FUNCTION_BLOCK AGVController (* Tamplate for a simple Basic Function Block Type *)
  (* Standard: 61499-2 *)
  (* Version 0.0, 2018-06-08, 4DIAC-IDE, 4DIAC-Consortium *)
  (* Version 1.0, 2016-05-26, AZ, fortiss GmbH *)
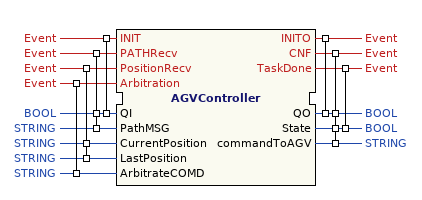
  EVENT_INPUT
    INIT WITH QI; (* Initialization Request *)
    PATHRecv WITH QI, PathMSG; (* Normal Execution Request *)
    PositionRecv WITH CurrentPosition, LastPosition;
    Arbitration WITH ArbitrateCOMD;
  END_EVENT
  EVENT_OUTPUT
    INITO WITH QO; (* Initialization Confirm *)
    CNF WITH QO, State, commandToAGV; (* Execution Confirmation *)
    TaskDone WITH State;
  END_EVENT
  VAR_INPUT
    QI : BOOL; (* Input event qualifier *)
    PathMSG : STRING; (* like 1-->3-.... *)
    CurrentPosition : STRING;
    LastPosition : STRING;
    ArbitrateCOMD : STRING;
  END_VAR
  VAR_OUTPUT
    QO : BOOL; (* Output event qualifier *)
    State : BOOL; (* busy or idle *)
    commandToAGV : STRING;
  END_VAR
  VAR
    ArbitrateCommand : BOOL := 0; (* Internal Variable *)
  END_VAR
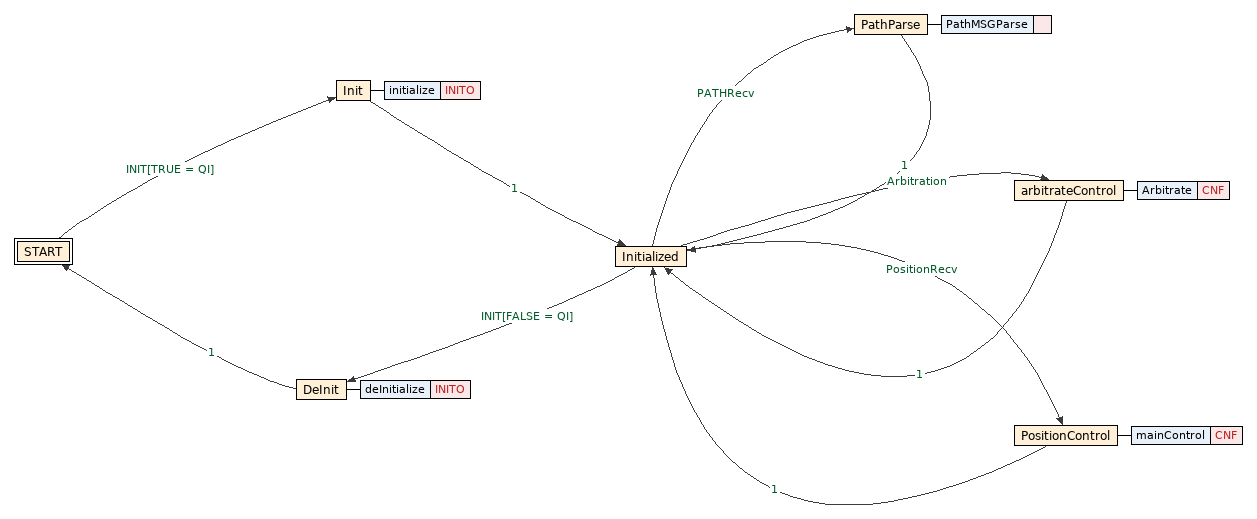
  EC_STATES
    START; (* Initial State *)
    Init : initialize -> INITO; (* Initialization *)
    PathParse : PathMSGParse; (* Normal execution *)
    Initialized;
    DeInit : deInitialize -> INITO;
    arbitrateControl : Arbitrate -> CNF;
    PositionControl : mainControl -> CNF;
  END_STATES
  EC_TRANSITIONS
    START TO Init := INIT[TRUE = QI];
    Init TO Initialized := 1;
    Initialized TO PathParse := PATHRecv;
    PathParse TO Initialized := 1;
    DeInit TO START := 1;
    Initialized TO DeInit := INIT[FALSE = QI];
    Initialized TO arbitrateControl := Arbitration;
    arbitrateControl TO Initialized := 1;
    Initialized TO PositionControl := PositionRecv;
    PositionControl TO Initialized := 1;
  END_TRANSITIONS
  ALGORITHM initialize IN ST: (* Initialization algorithm *)
QO := QI;
  END_ALGORITHM
  ALGORITHM deInitialize IN ST: (* Normally executed algorithm *)
QO := FALSE;
  END_ALGORITHM
  ALGORITHM PathMSGParse IN ST: (* new algorithm *)
QO := QI;

IF TRUE  = QI THEN
  (*  only perform normal operation of QI is true*)

END_IF;
  END_ALGORITHM
  ALGORITHM Arbitrate IN ST: (* new algorithm *)

  END_ALGORITHM
  ALGORITHM mainControl IN ST: (* new algorithm *)

  END_ALGORITHM
END_FUNCTION_BLOCK
